// TIA Portal V20 export
TYPE "LDrvSafe_typeSinaTlg903Status"
TITLE = LDrvSafe_typeSinaTlg903Status
// Failsafe user-defined data type for PROFIsafe telegram 903 to get status information of Safety Integrated Functions of SINAMICS
// stored: IsFailsafeCompliant true
   STRUCT
      STOactive { ExternalWritable := 'False'} : Bool;   // Safety Function Safe Torque Off active
      SS1active { ExternalWritable := 'False'} : Bool;   // Safety Function Safe Stop 1 active
      SS2active { ExternalWritable := 'False'} : Bool;   // Safety Function Safe Stop 2 active
      SOSactive { ExternalWritable := 'False'} : Bool;   // Safety Function Safe Operating Stop active
      SLSactive { ExternalWritable := 'False'} : Bool;   // Safety Function Safely-limited Speed active
      reserved1 { ExternalWritable := 'False'} : Bool;   // Reserve bit 1
      SLPactive { ExternalWritable := 'False'} : Bool;   // Safety Function Safely-limited Position active
      internalEvent { ExternalWritable := 'False'} : Bool;   // Internal Event occured (Safety error in SINAMICS)
      SLAactive { ExternalWritable := 'False'} : Bool;   // Safety Function Safely-limited Acceleration active
      SLSbit0Active { ExternalWritable := 'False'} : Bool;   // One of the the four SLS limits is active; operates together with bit 1
      SLSbit1Active { ExternalWritable := 'False'} : Bool;   // One of the the four SLS limits is active; operates together with bit 0
      reserved3 { ExternalWritable := 'False'} : Bool;   // Reserve bit 3
      SDIpositiveActive { ExternalWritable := 'False'} : Bool;   // Safety Function Safe Direction (positive direction) active
      SDInegativeActive { ExternalWritable := 'False'} : Bool;   // Safety Function Safe Direction (negative direction) active
      reserved4 { ExternalWritable := 'False'} : Bool;   // Reserve bit 4
      SSMactive { ExternalWritable := 'False'} : Bool;   // Safety Function Safe Speed Monitor; signals, if safe speed is below paramterizable speed limit
      reserved5 { ExternalWritable := 'False'} : Bool;   // Reserve bit 5
      reserved6 { ExternalWritable := 'False'} : Bool;   // Reserve bit 6
      reserved7 { ExternalWritable := 'False'} : Bool;   // Reserve bit 7
      SLPrangeActive { ExternalWritable := 'False'} : Bool;   // SLP position range 1 or 2 is active
      reserved8 { ExternalWritable := 'False'} : Bool;   // Reserve bit 8
      reserved9 { ExternalWritable := 'False'} : Bool;   // Reserve bit 9
      safePositionValid { ExternalWritable := 'False'} : Bool;   // Safe Position is valid
      safelyReferenced { ExternalWritable := 'False'} : Bool;   // Drive is safely referenced
      statusFDI0 { ExternalWritable := 'False'} : Bool;   // Status of Failsafe Digital Input 0
      statusFDI1 { ExternalWritable := 'False'} : Bool;   // Status of Failsafe Digital Input 1
      statusFDI2 { ExternalWritable := 'False'} : Bool;   // Status of Failsafe Digital Input 2
      SS2ESRactive { ExternalWritable := 'False'} : Bool;   // Safety Function SS2ESR active
      SS2Eactive { ExternalWritable := 'False'} : Bool;   // Safety Function SS2E active
      SOSselected { ExternalWritable := 'False'} : Bool;   // Safety Function Safe Operating Stop selected (not active yet)
      SLPupperLimitMaintained { ExternalWritable := 'False'} : Bool;   // SLP: upper limit maintained
      SLPlowerLimitMaintained { ExternalWritable := 'False'} : Bool;   // SLP: lower limit maintained
      SCA1 { ExternalWritable := 'False'} : Bool;   // Safe Cam 1
      SCA2 { ExternalWritable := 'False'} : Bool;   // Safe Cam 2
      SCA3 { ExternalWritable := 'False'} : Bool;   // Safe Cam 3
      SCA4 { ExternalWritable := 'False'} : Bool;   // Safe Cam 4
      SCA5 { ExternalWritable := 'False'} : Bool;   // Safe Cam 5
      SCA6 { ExternalWritable := 'False'} : Bool;   // Safe Cam 6
      SCA7 { ExternalWritable := 'False'} : Bool;   // Safe Cam 7
      SCA8 { ExternalWritable := 'False'} : Bool;   // Safe Cam 8
      SCA9 { ExternalWritable := 'False'} : Bool;   // Safe Cam 9
      SCA10 { ExternalWritable := 'False'} : Bool;   // Safe Cam 10
      SCA11 { ExternalWritable := 'False'} : Bool;   // Safe Cam 11
      SCA12 { ExternalWritable := 'False'} : Bool;   // Safe Cam 12
      SCA13 { ExternalWritable := 'False'} : Bool;   // Safe Cam 13
      SCA14 { ExternalWritable := 'False'} : Bool;   // Safe Cam 14
      SCA15 { ExternalWritable := 'False'} : Bool;   // Safe Cam 15
      SCA16 { ExternalWritable := 'False'} : Bool;   // Safe Cam 16
      SCA17 { ExternalWritable := 'False'} : Bool;   // Safe Cam 17
      SCA18 { ExternalWritable := 'False'} : Bool;   // Safe Cam 18
      SCA19 { ExternalWritable := 'False'} : Bool;   // Safe Cam 19
      SCA20 { ExternalWritable := 'False'} : Bool;   // Safe Cam 20
      SCA21 { ExternalWritable := 'False'} : Bool;   // Safe Cam 21
      SCA22 { ExternalWritable := 'False'} : Bool;   // Safe Cam 22
      SCA23 { ExternalWritable := 'False'} : Bool;   // Safe Cam 23
      SCA24 { ExternalWritable := 'False'} : Bool;   // Safe Cam 24
      SCA25 { ExternalWritable := 'False'} : Bool;   // Safe Cam 25
      SCA26 { ExternalWritable := 'False'} : Bool;   // Safe Cam 26
      SCA27 { ExternalWritable := 'False'} : Bool;   // Safe Cam 27
      SCA28 { ExternalWritable := 'False'} : Bool;   // Safe Cam 28
      SCA29 { ExternalWritable := 'False'} : Bool;   // Safe Cam 29
      SCA30 { ExternalWritable := 'False'} : Bool;   // Safe Cam 30
      SCAactive { ExternalWritable := 'False'} : Bool;   // Safety Function Safe Cam active
      SCAvalid { ExternalWritable := 'False'} : Bool;   // Safety Function Safe Cam valid
      variableSLSvalue { ExternalWritable := 'False'} : Int;   // Actual SLS value for SLS limit 1
   END_STRUCT;
END_TYPE
